FUNCTION F_StateEnumToString : STRING
VAR_INPUT
	eState : eSingleState;
END_VAR
VAR
END_VAR

CASE eState OF
    eSingleState.Idle:
        F_StateEnumToString := 'Idle';
    eSingleState.Execute:
        F_StateEnumToString := 'Execute';
    eSingleState.Stopping:
        F_StateEnumToString := 'Stopping';
    eSingleState.Stopped:
        F_StateEnumToString := 'Stopped';
    eSingleState.Suspending:
        F_StateEnumToString := 'Suspending';
    eSingleState.Suspended:
        F_StateEnumToString := 'Suspended';
    eSingleState.Aborting:
        F_StateEnumToString := 'Aborting';
    eSingleState.Aborted:
        F_StateEnumToString := 'Aborted';
ELSE
    F_StateEnumToString := 'Unknown';
END_CASE

END_FUNCTION

(* stored: Version 1.1.0.1
   POU F_StateEnumToString: Id {938c23a4-80a0-4d0f-af13-e5917da633ac}, SpecialFunc None *)
